FUNCTION_BLOCK PUBLIC CommandBase IMPLEMENTS ICommand
VAR_INPUT
END_VAR
VAR_IN_OUT
END_VAR
VAR
	_execute		: BOOL;		// Wird von PCS gesetzt um die Ausführung zu starten; zurücksetzen bricht die Ausführung ab
	_busy			: BOOL;		// Anzeige, dass die Ausführung in der SPS läuft
	_ResultCode		: UINT;		// Resultat der letzten Ausführung (bExecute & bBusy = FALSE)
	counter: UINT;
END_VAR

// OO-Class 
;

// Stops execution of Command 
METHOD PUBLIC Abort
Execute := FALSE;
Busy := FALSE;
ResultCode := 5; // canceled
END_METHOD

//Anzeige, dass die Ausführung in der SPS läuft
{attribute 'monitoring' := 'variable'}
PROPERTY PUBLIC Busy : BOOL
GET // PUBLIC
Busy := _busy;
END_GET
SET // Protected
_busy := Busy;
END_SET
END_PROPERTY

METHOD PROTECTED Done
ResultCode := 0; // done
Execute := FALSE;
Busy := FALSE;
END_METHOD

// Wird von PCS gesetzt um die Ausführung zu starten; zurücksetzen bricht die Ausführung ab
{attribute 'monitoring' := 'call'}
PROPERTY PUBLIC Execute : BOOL
GET // PUBLIC
Execute := _execute;
END_GET
SET // PUBLIC
_execute := Execute;
END_SET
END_PROPERTY

// Update the state of the command button. Should be called every cycle.
METHOD PUBLIC Refresh
VAR_INPUT
END_VAR
counter := counter + 1;

// Länger gehendes Kommando
IF Execute THEN
	Busy := TRUE;
END_IF

// Reset Case
IF NOT Execute AND Busy THEN
	// Abort
	Abort();
END_IF

IF Execute AND Busy THEN
	ResultCode := 4; // running
	IF Task() THEN
		Done();
	END_IF
END_IF
END_METHOD

// Resultat der letzten Ausführung (bExecute & bBusy = FALSE)
{attribute 'monitoring' := 'variable'}
PROPERTY ResultCode : UINT
GET // PUBLIC
ResultCode := _resultCode;
END_GET
SET // PROTECTED
_resultCode := ResultCode;
END_SET
END_PROPERTY

// Execute the funktional part of the command implementation
METHOD PROTECTED Task : BOOL
;
END_METHOD

END_FUNCTION_BLOCK

(* stored: Version 1.1.0.1, ProductVersion 3.1.4022.10
   POU CommandBase: Id {5ed0d5bd-0ff5-4097-ae74-31498bed2e22}, SpecialFunc None
   Method Abort: Id {b3999881-28f7-422e-bf1b-eba84960aef3}
   Property Busy: Id {f17dea9b-0491-471d-bdd6-8776e5a75cd7}
   Get Get: Id {15f9358f-22b9-461b-8c58-f932ab10aac1}
   Set Set: Id {21101625-0a3e-4ca4-939b-729925182e47}
   Method Done: Id {e44fa825-a28e-46f6-bd9b-b7a6061e20a7}
   Property Execute: Id {f9d7f224-aeca-4a8d-b244-62b6043700af}
   Get Get: Id {07b42bf6-49a9-48fb-a416-3adb67c85587}
   Set Set: Id {f18849aa-ced1-409e-9b14-6534753dab53}
   Method Refresh: Id {8e66b5e0-e08f-4024-b1ed-2b1412f1580f}
   Property ResultCode: Id {ac5fe93e-2c3e-4e72-a2f6-add14726c137}
   Get Get: Id {b127a023-a4b1-4a5b-90fc-f47fb8009b3a}
   Set Set: Id {c03ce2dd-ce5f-4dcf-b315-9a5df15e8650}
   Method Task: Id {6e407172-b849-400a-8c24-c3a1ccb62b55} *)
